INTERFACE I_Cycle EXTENDS I_Object

METHOD PUBLIC M_Cycle
VAR_INPUT
END_VAR
END_METHOD

END_INTERFACE

(* stored: Version 1.1.0.1
   Itf I_Cycle: Id {525606fa-ed43-0c71-29bd-f72b8f0a0b08}
   Method M_Cycle: Id {fb8f04cf-e108-0b45-279b-00e8a36dafa3} *)
